{attribute 'qualified_only'}
{attribute 'strict'}
{attribute 'to_string'}
TYPE eObjectSensorState :
(
	AUS 					:= 0,				// Das Objekt ist ausgeschalten
	LAUFEND 				:= 1,				// Das Objekt ist aktiv
	FEHLER					:= 2				// Es gibt einen Fehler bezüglich des Objektes
);
END_TYPE

(* stored: Version 1.1.0.1
   DUT eObjectSensorState: Id {dbbc4957-3eda-4333-800c-8a51ebe3ba0a} *)
